ORGANIZATION_BLOCK 主程序:OB1
TITLE=程序注释
BEGIN
Network 1 // 网络标题
// 网络注释
LD     I0.0
LD     I0.1
CTD    C20, +3
Network 2
LD     C20
=      Q0.0
END_ORGANIZATION_BLOCK
SUBROUTINE_BLOCK SBR_0:SBR0
TITLE=子程序注释
BEGIN
Network 1 // 网络标题
// 网络注释
END_SUBROUTINE_BLOCK
INTERRUPT_BLOCK INT_0:INT0
TITLE=中断程序注释
BEGIN
Network 1 // 网络标题
// 网络注释
END_INTERRUPT_BLOCK
